// TIA Portal V17 export
// export: Created 2025-05-22T06:01:23.9340658Z, ExportSetting WithDefaults, DisplayName Totally Integrated Automation Portal, DisplayVersion V17 Update 8, DisplayName TIA Portal Openness, DisplayVersion V17 Update 8, DisplayName TIA Portal Version Control Interface, DisplayVersion V17, DisplayName SINAMICS Startdrive Advanced, DisplayVersion V17 SP2, DisplayName SINAMICS Startdrive G110M, G120, G120C, G120D, G120P, G115D, DisplayVersion V17 SP2, DisplayName SINAMICS Startdrive G130, G150, S120, S150, SINAMICS MV, S210, DisplayVersion V17 SP2, DisplayName STEP 7 Professional, DisplayVersion V17 Update 8, DisplayName SINUMERIK ONE STEP 7 Toolbox, DisplayVersion V17 Update 12, DisplayName SINUMERIK ONE PLC Basic Program Plus, DisplayVersion V17 Update 12, DisplayName SINUMERIK 840D sl STEP 7 Toolbox, DisplayVersion V17 Update 12, DisplayName STEP 7 Safety, DisplayVersion V17 Update 6, DisplayName WinCC Advanced, DisplayVersion V17 Update 8
DATA_BLOCK "DB7263_UNIT_1_LASER_ENABLE_DISABLE"   // DB7263
AUTHOR : ETXETAR
VERSION : 1.0
// stored: AutoNumber false, DBAccessibleFromOPCUA true, DBAccessibleFromWebserver true, InstanceOfName FB7255_ENABLE_DISABLE, InstanceOfType FB
"FB7255_ENABLE_DISABLE"
   // VAR_INPUT
   //    OPTIONS_0 : Byte;
   //    ENABLE_CONDITIONS_I : Bool;
   //    DISABLE_CONDITIONS_I : Bool;
   //    ENABLE_DISABLE_LINE_REQUEST : Int;
   //    DISABLE_WITH : Bool;
   //    ENABLE_WITH : Bool;
   //    HW_DEVICE : HW_DEVICE;
   // END_VAR
   // VAR_OUTPUT
   //    ENABLED : Bool;
   //    DISABLED : Bool;
   //    DISABLED_WARNING : Bool;
   // END_VAR
   // VAR RETAIN
   //    ENABLE_CONDITIONS : Bool;
   //    DISABLE_CONDITIONS : Bool;
   //    ENABLE_REQUEST : Bool;
   //    DISABLE_REQUEST : Bool;
   //    WARNING_GONE : Bool;
   //    PULSE_1 : Bool;
   //    PREVIOUS_ENABLE_STATE : Bool;
   //    DISABLE_ENABLE_REQUEST : Bool;
   //    MODE_DIS_ENABLE : Byte;
   // END_VAR
BEGIN
END_DATA_BLOCK
